(* PLC project Unnamed, Unknown Unnamed 1 *)
(* stored: creationDateTime 2023-03-10T10:37:17, modificationDateTime 2023-03-15T15:56:42 *)

(* 978-3-658-16137-8, p.168 *)
FUNCTION_BLOCK Antivalence_3x
  VAR_INPUT
    IN0 : BOOL;
    IN1 : BOOL;
    IN2 : BOOL;
  END_VAR
  VAR_OUTPUT
    OUT1 : BOOL;
  END_VAR

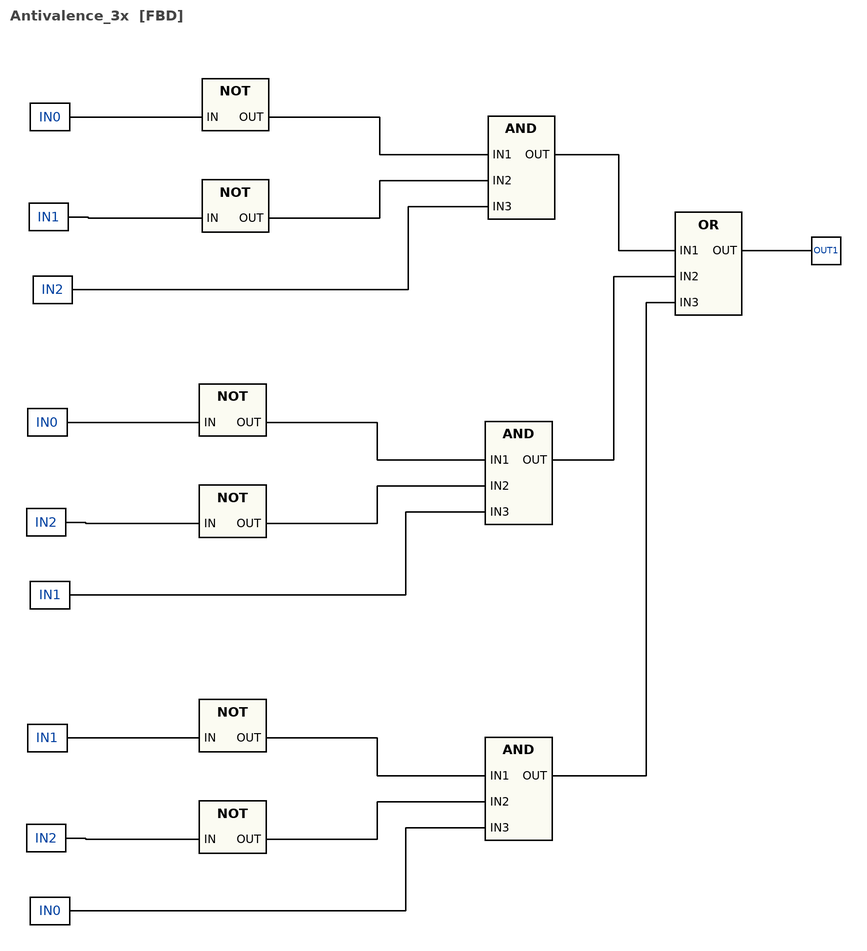
(* FBD diagram, written out as Structured Text *)
OUT1 := NOT IN0 AND NOT IN1 AND IN2 OR NOT IN0 AND NOT IN2 AND IN1 OR NOT IN1 AND NOT IN2 AND IN0;
END_FUNCTION_BLOCK

CONFIGURATION config
  RESOURCE resource1 ON PLC
  END_RESOURCE
END_CONFIGURATION
